(* IEC 61131-3 sources: Summary-ETFA22/benchmark/PLCopen_safety (part 2) *)

(* ---- SFOutControl.st ---- *)
PROGRAM Main
VAR_INPUT
    Activate : BOOL ;
    SSafeControl : SAFEBOOL ;
    ProcessControl : BOOL ;
    StaticControl : BOOL ;
    SStartReset : SAFEBOOL ;
    SAutoReset	: SAFEBOOL ;
    Reset : BOOL ;
END_VAR
VAR
    SFOutControl : SFOutControl;
END_VAR
SFOutControl(Activate:=Activate,SSafeControl:=SSafeControl,ProcessControl:=ProcessControl,StaticControl:=StaticControl,
SStartReset:=SStartReset,SAutoReset:=SAutoReset,Reset:=Reset);
END_PROGRAM

FUNCTION_BLOCK SFOutControl
VAR_INPUT
    Activate : BOOL ;
    SSafeControl : SAFEBOOL ;
    ProcessControl : BOOL ;
    StaticControl : BOOL ;
    SStartReset : SAFEBOOL ;
    SAutoReset	: SAFEBOOL ;
    Reset : BOOL ;
END_VAR
VAR
    RTRIGatResetQ : BOOL;
    RTRIGatResetM : BOOL;
    RTRIGatProcessControlQ : BOOL;
    RTRIGatProcessControlM : BOOL;
END_VAR
VAR_OUTPUT
    Ready : BOOL ;
    SOutControl : SAFEBOOL ;
    Error : BOOL ;
    DiagCode : WORD:=16#0000 ;
END_VAR
RTRIGatResetQ := Reset AND NOT RTRIGatResetM;
RTRIGatResetM := Reset;

RTRIGatProcessControlQ := ProcessControl AND NOT RTRIGatProcessControlM;
RTRIGatProcessControlM := ProcessControl;

IF NOT Activate THEN
    DiagCode := 16#0000;
ELSE
    CASE DiagCode OF
    16#0000:
        IF Activate THEN
            DiagCode := 16#8001;
        END_IF;
    16#8000:
        IF NOT SSafeControl THEN
            DiagCode := 16#8002;
        ELSIF NOT ProcessControl THEN
            DiagCode := 16#8010;
        END_IF;
    16#8001:
        IF Reset AND NOT RTRIGatResetQ AND NOT SStartReset THEN
            DiagCode := 16#C001;
        ELSIF RTRIGatResetQ AND RTRIGatProcessControlQ THEN
            DiagCode := 16#C111;
        ELSIF RTRIGatResetQ OR SStartReset THEN
            DiagCode := 16#8010;
        END_IF;
    16#8002:
        IF SSafeControl THEN
            DiagCode := 16#8003;
        END_IF;
    16#8003:
        IF NOT SSafeControl THEN
            DiagCode := 16#8002;
        ELSIF Reset AND NOT RTRIGatResetQ AND NOT SAutoReset THEN
            DiagCode := 16#C002;
        ELSIF RTRIGatResetQ AND RTRIGatProcessControlQ THEN
            DiagCode := 16#C211;
        ELSIF RTRIGatResetQ OR SAutoReset THEN
            DiagCode := 16#8010;
        END_IF;
    16#8010:
        IF NOT SSafeControl THEN
            DiagCode := 16#8002;
        ELSIF NOT RTRIGatProcessControlQ AND ProcessControl AND NOT StaticControl THEN
            DiagCode := 16#C010;
        ELSIF SSafeControl AND (RTRIGatProcessControlQ OR (StaticControl AND ProcessControl)) THEN
            DiagCode := 16#8000;
        END_IF;
    16#C001:
        IF NOT Reset THEN
            DiagCode := 16#8001;
        END_IF;
    16#C002:
        IF NOT Reset THEN
            DiagCode := 16#8003;
        END_IF;
    16#C010:
        IF NOT ProcessControl THEN
            DiagCode := 16#8010;
        END_IF;
    16#C111:
        IF NOT Reset THEN
            DiagCode := 16#8001;
        END_IF;
    16#C211:
        IF NOT Reset THEN
            DiagCode := 16#8003;
        END_IF;
    END_CASE;
END_IF;
CASE DiagCode OF
16#0000:
    Ready := FALSE;
    SOutControl := FALSE;
    Error := FALSE;
16#8000:
    Ready := TRUE;
    SOutControl := TRUE;
    Error := FALSE;
16#8001, 16#8002, 16#8003, 16#8010:
    Ready := TRUE;
    SOutControl := FALSE;
    Error := FALSE;
16#C001, 16#C002, 16#C010, 16#C111, 16#C211:
    Ready := TRUE;
    SOutControl := FALSE;
    Error := TRUE;
END_CASE;
END_FUNCTION_BLOCK

(* ---- SFOutControl_CAP.st ---- *)
PROGRAM Main
VAR_INPUT
    Activate : BOOL ;
    SSafeControl : SAFEBOOL ;
    ProcessControl : BOOL ;
    StaticControl : BOOL ;
    SStartReset : SAFEBOOL ;
    SAutoReset	: SAFEBOOL ;
    Reset : BOOL ;
END_VAR
VAR
    SFOutControl : SFOutControl;
END_VAR
SFOutControl(Activate:=Activate,SSafeControl:=SSafeControl,ProcessControl:=ProcessControl,StaticControl:=StaticControl,
SStartReset:=SStartReset,SAutoReset:=SAutoReset,Reset:=Reset);
END_PROGRAM

FUNCTION_BLOCK SFOutControl
VAR_INPUT
    Activate : BOOL ;
    SSafeControl : SAFEBOOL ;
    ProcessControl : BOOL ;
    StaticControl : BOOL ;
    SStartReset : SAFEBOOL ;
    SAutoReset	: SAFEBOOL ;
    Reset : BOOL ;
END_VAR
VAR
    RTRIGatResetQ : BOOL;
    RTRIGatResetM : BOOL;
    RTRIGatProcessControlQ : BOOL;
    RTRIGatProcessControlM : BOOL;
END_VAR
VAR_OUTPUT
    Ready : BOOL ;
    SOutControl : SAFEBOOL ;
    Error : BOOL ;
    DiagCode : WORD:=16#0000 ;
END_VAR
RTRIGatResetQ := Reset AND NOT RTRIGatResetM;
RTRIGatResetM := Reset;

RTRIGatProcessControlQ := ProcessControl AND NOT RTRIGatProcessControlM;
RTRIGatProcessControlM := ProcessControl;

IF NOT Activate THEN
    DiagCode := change(16#0000, 16#0000);
ELSE
    CASE DiagCode OF
    16#0000:
        IF Activate THEN
            DiagCode := 16#8001;
        END_IF;
    16#8000:
        IF NOT SSafeControl THEN
            DiagCode := 16#8002;
        ELSIF NOT ProcessControl THEN
            DiagCode := 16#8010;
        END_IF;
    16#8001:
        IF Reset AND NOT RTRIGatResetQ AND NOT SStartReset THEN
            DiagCode := 16#C001;
        ELSIF RTRIGatResetQ AND RTRIGatProcessControlQ THEN
            DiagCode := 16#C111;
        ELSIF RTRIGatResetQ OR SStartReset THEN
            DiagCode := 16#8010;
        END_IF;
    16#8002:
        IF SSafeControl THEN
            DiagCode := 16#8003;
        END_IF;
    16#8003:
        IF NOT SSafeControl THEN
            DiagCode := 16#8002;
        ELSIF Reset AND NOT RTRIGatResetQ AND NOT SAutoReset THEN
            DiagCode := 16#C002;
        ELSIF RTRIGatResetQ AND RTRIGatProcessControlQ THEN
            DiagCode := 16#C211;
        ELSIF RTRIGatResetQ OR SAutoReset THEN
            DiagCode := 16#8010;
        END_IF;
    16#8010:
        IF NOT SSafeControl THEN
            DiagCode := 16#8002;
        ELSIF NOT RTRIGatProcessControlQ AND ProcessControl AND NOT StaticControl THEN
            DiagCode := 16#C010;
        ELSIF SSafeControl AND (RTRIGatProcessControlQ OR (StaticControl AND ProcessControl)) THEN
            DiagCode := 16#8000;
        END_IF;
    16#C001:
        IF NOT Reset THEN
            DiagCode := change(16#8001, 16#C002);
        END_IF;
    16#C002:
        IF NOT Reset THEN
            DiagCode := 16#8003;
        END_IF;
    16#C010:
        IF NOT ProcessControl THEN
            DiagCode := 16#8010;
        END_IF;
    16#C111:
        IF NOT Reset THEN
            DiagCode := 16#8001;
        END_IF;
    16#C211:
        IF NOT Reset THEN
            DiagCode := 16#8003;
        END_IF;
    END_CASE;
END_IF;
CASE DiagCode OF
16#0000:
    Ready := FALSE;
    SOutControl := FALSE;
    Error := FALSE;
16#8000:
    Ready := TRUE;
    SOutControl := TRUE;
    Error := FALSE;
16#8001, 16#8002, 16#8003, 16#8010:
    Ready := TRUE;
    SOutControl := FALSE;
    Error := FALSE;
16#C001, 16#C002, 16#C010, 16#C111, 16#C211:
    Ready := TRUE;
    SOutControl := FALSE;
    Error := TRUE;
END_CASE;
END_FUNCTION_BLOCK

(* ---- SFSafelyLimitSpeed.st ---- *)
PROGRAM Main
VAR_INPUT
    Activate : BOOL;
    SOpMode : SAFEBOOL;
    SEnabled : SAFEBOOL;
    AxisID : INT;
    MonitoringTime : TIME;
    Reset : BOOL;
    Acknowledge : BOOL;      (* This is an internal input *)
END_VAR
VAR
    SFSafelyLimitSpeed : SFSafelyLimitSpeed;
END_VAR
SFSafelyLimitSpeed(Activate:=Activate,SOpMode:=SOpMode,SEnabled:=SEnabled,AxisID:=AxisID,MonitoringTime:=MonitoringTime,
Reset:=Reset,Acknowledge:=Acknowledge);
END_PROGRAM

FUNCTION_BLOCK SFSafelyLimitSpeed
VAR_INPUT
    Activate : BOOL;
    SOpMode : SAFEBOOL;
    SEnabled : SAFEBOOL;
    AxisID : INT;
    MonitoringTime : TIME;
    Reset : BOOL;
    Acknowledge : BOOL;      (* This is an internal input *)
END_VAR
VAR
    IN : BOOL;
    PT : TIME;
    running : BOOL;
    Q : BOOL;
    RTRIGatResetQ : BOOL;
    RTRIGatResetM : BOOL;
END_VAR
VAR_OUTPUT
    Ready : BOOL;
    SSafetyActive : SAFEBOOL;
    Error : BOOL;
    DiagCode : WORD;
END_VAR
RTRIGatResetQ := Reset AND NOT RTRIGatResetM;
RTRIGatResetM := Reset;

IF NOT Activate THEN
    DiagCode := 16#0000;
END_IF;
IN:=Activate AND NOT SOpMode;
PT:=MonitoringTime;
IF NOT IN THEN
    Q := FALSE;
    running := FALSE;
ELSIF NOT running AND NOT Q THEN
    running := TRUE;
ELSIF running AND NOT Q THEN
    Q := NONDETERMINISTIC_BOOL();
    running := NOT Q;
END_IF;
CASE DiagCode OF
16#0000:
    IF Activate THEN
        DiagCode := 16#8001;
    END_IF;
16#8000:
    IF NOT Acknowledge THEN
        DiagCode := 16#C002;
    ELSIF SOpMode THEN
        DiagCode := 16#8012;
    ELSIF SEnabled THEN
        DiagCode := 16#8004;
    END_IF;
16#8001:
    IF Reset AND NOT RTRIGatResetQ THEN
        DiagCode := 16#C001;
    ELSIF RTRIGatResetQ AND NOT Acknowledge THEN
        DiagCode := 16#8002;
    ELSIF RTRIGatResetQ AND Acknowledge THEN
        DiagCode := 16#8012;
    END_IF;
16#8002:
    IF NOT SOpMode THEN
        DiagCode := 16#8003;
    ELSIF Acknowledge THEN
        DiagCode := 16#8012;
    END_IF;
16#8003:
    IF Q THEN
        DiagCode := 16#C003;
    ELSIF SOpMode THEN
        DiagCode := 16#8012;
    ELSIF Acknowledge AND NOT SEnabled THEN
        DiagCode := 16#8000;
    ELSIF Acknowledge AND SEnabled THEN
        DiagCode := 16#8004;
    END_IF;
16#8004:
    IF NOT Acknowledge THEN
        DiagCode := 16#C002;
    ELSIF SOpMode THEN
        DiagCode := 16#8012;
    ELSIF NOT SEnabled THEN
        DiagCode := 16#8000;
    END_IF;
16#8005:
    IF SOpMode THEN
        DiagCode := 16#8012;
    END_IF;
16#8012:
    IF NOT Acknowledge THEN
        DiagCode := 16#8002;
    ELSIF NOT SOpMode THEN
        DiagCode := 16#8003;
    END_IF;
16#C001:
    IF NOT Reset THEN
        DiagCode := 16#8001;
    END_IF;
16#C002:
    IF Reset AND NOT RTRIGatResetQ THEN
        DiagCode := 16#C004;
    ELSIF RTRIGatResetQ THEN
        DiagCode := 16#8005;
    END_IF;
16#C003:
    IF Reset AND NOT RTRIGatResetQ THEN
        DiagCode := 16#C005;
    ELSIF RTRIGatResetQ THEN
        DiagCode := 16#8005;
    END_IF;
16#C004:
    IF NOT Reset THEN
        DiagCode := 16#C002;
    END_IF;
16#C005:
    IF NOT Reset THEN
        DiagCode := 16#C003;
    END_IF;
END_CASE;
CASE DiagCode OF
16#0000:
    Ready := FALSE;
    SSafetyActive := FALSE;
    Error := FALSE;
16#8000,
16#8004:
    Ready := TRUE;
    SSafetyActive := TRUE;
    Error := FALSE;
16#8001,
16#8002,
16#8003,
16#8005,
16#8012:
    Ready := TRUE;
    SSafetyActive := FALSE;
    Error := FALSE;
16#C001,
16#C002,
16#C003,
16#C004,
16#C005:
    Ready := TRUE;
    SSafetyActive := FALSE;
    Error := TRUE;
END_CASE;
END_FUNCTION_BLOCK

(* ---- SFSafelyLimitSpeed_CAP.st ---- *)
PROGRAM Main
VAR_INPUT
    Activate : BOOL;
    SOpMode : SAFEBOOL;
    SEnabled : SAFEBOOL;
    AxisID : INT;
    MonitoringTime : TIME;
    Reset : BOOL;
    Acknowledge : BOOL;      (* This is an internal input *)
END_VAR
VAR
    SFSafelyLimitSpeed : SFSafelyLimitSpeed;
END_VAR
SFSafelyLimitSpeed(Activate:=Activate,SOpMode:=SOpMode,SEnabled:=SEnabled,AxisID:=AxisID,MonitoringTime:=MonitoringTime,
Reset:=Reset,Acknowledge:=Acknowledge);
END_PROGRAM

FUNCTION_BLOCK SFSafelyLimitSpeed
VAR_INPUT
    Activate : BOOL;
    SOpMode : SAFEBOOL;
    SEnabled : SAFEBOOL;
    AxisID : INT;
    MonitoringTime : TIME;
    Reset : BOOL;
    Acknowledge : BOOL;      (* This is an internal input *)
END_VAR
VAR
    IN : BOOL;
    PT : TIME;
    running : BOOL;
    Q : BOOL;
    RTRIGatResetQ : BOOL;
    RTRIGatResetM : BOOL;
END_VAR
VAR_OUTPUT
    Ready : BOOL;
    SSafetyActive : SAFEBOOL;
    Error : BOOL;
    DiagCode : WORD;
END_VAR
RTRIGatResetQ := Reset AND NOT RTRIGatResetM;
RTRIGatResetM := Reset;

IF NOT Activate THEN
    DiagCode := 16#0000;
END_IF;
IN:=Activate AND NOT SOpMode;
PT:=MonitoringTime;
IF NOT IN THEN
    Q := FALSE;
    running := FALSE;
ELSIF NOT running AND NOT Q THEN
    running := TRUE;
ELSIF running AND NOT Q THEN
    Q := NONDETERMINISTIC_BOOL();
    running := NOT Q;
END_IF;
CASE DiagCode OF
16#0000:
    IF Activate THEN
        DiagCode := 16#8001;
    END_IF;
16#8000:
    IF NOT Acknowledge THEN
        DiagCode := change(16#C002, 16#8012);
    ELSIF SOpMode THEN
        DiagCode := 16#8012;
    ELSIF SEnabled THEN
        DiagCode := 16#8004;
    END_IF;
16#8001:
    IF Reset AND NOT RTRIGatResetQ THEN
        DiagCode := 16#C001;
    ELSIF RTRIGatResetQ AND NOT Acknowledge THEN
        DiagCode := 16#8002;
    ELSIF RTRIGatResetQ AND Acknowledge THEN
        DiagCode := 16#8012;
    END_IF;
16#8002:
    IF NOT SOpMode THEN
        DiagCode := 16#8003;
    ELSIF Acknowledge THEN
        DiagCode := 16#8012;
    END_IF;
16#8003:
    IF Q THEN
        DiagCode := 16#C003;
    ELSIF SOpMode THEN
        DiagCode := 16#8012;
    ELSIF Acknowledge AND NOT SEnabled THEN
        DiagCode := 16#8000;
    ELSIF Acknowledge AND SEnabled THEN
        DiagCode := 16#8004;
    END_IF;
16#8004:
    IF NOT Acknowledge THEN
        DiagCode := 16#C002;
    ELSIF SOpMode THEN
        DiagCode := 16#8012;
    ELSIF NOT SEnabled THEN
        DiagCode := 16#8000;
    END_IF;
16#8005:
    IF SOpMode THEN
        DiagCode := 16#8012;
    END_IF;
16#8012:
    IF NOT Acknowledge THEN
        DiagCode := 16#8002;
    ELSIF NOT SOpMode THEN
        DiagCode := 16#8003;
    END_IF;
16#C001:
    IF NOT Reset THEN
        DiagCode := 16#8001;
    END_IF;
16#C002:
    IF Reset AND NOT RTRIGatResetQ THEN
        DiagCode := 16#C004;
    ELSIF RTRIGatResetQ THEN
        DiagCode := 16#8005;
    END_IF;
16#C003:
    IF Reset AND NOT RTRIGatResetQ THEN
        DiagCode := 16#C005;
    ELSIF RTRIGatResetQ THEN
        DiagCode := 16#8005;
    END_IF;
16#C004:
    IF NOT Reset THEN
        DiagCode := 16#C002;
    END_IF;
16#C005:
    IF NOT Reset THEN
        DiagCode := 16#C003;
    END_IF;
END_CASE;
CASE DiagCode OF
16#0000:
    Ready := FALSE;
    SSafetyActive := FALSE;
    Error := FALSE;
16#8000,
16#8004:
    Ready := TRUE;
    SSafetyActive := TRUE;
    Error := FALSE;
16#8001,
16#8002,
16#8003,
16#8005,
16#8012:
    Ready := TRUE;
    SSafetyActive := FALSE;
    Error := FALSE;
16#C001,
16#C002,
16#C003,
16#C004,
16#C005:
    Ready := TRUE;
    SSafetyActive := FALSE;
    Error := TRUE;
END_CASE;
END_FUNCTION_BLOCK

(* ---- SFSafeStop.st ---- *)
PROGRAM Main
VAR_INPUT
    Activate : BOOL;
    SStopIn : SAFEBOOL;
    AxisID : INT;
    MonitoringTime : TIME;
    Reset : BOOL;
    Acknowledge : BOOL;      (* This is an internal input *)
END_VAR
VAR
    SFSafeStop : SFSafeStop;
END_VAR
SFSafeStop(Activate:=Activate,SStopIn:=SStopIn,AxisID:=AxisID,MonitoringTime:=MonitoringTime,Reset:=Reset,
Acknowledge:=Acknowledge);
END_PROGRAM

FUNCTION_BLOCK SFSafeStop
VAR_INPUT
    Activate : BOOL;
    SStopIn : SAFEBOOL;
    AxisID : INT;
    MonitoringTime : TIME;
    Reset : BOOL;
    Acknowledge : BOOL;      (* This is an internal input *)
END_VAR
VAR
    IN : BOOL;
    PT : TIME;
    running : BOOL;
    Q : BOOL;
    RTRIGatResetQ : BOOL;
    RTRIGatResetM : BOOL;
END_VAR
VAR_OUTPUT
    Ready : BOOL;
    SStopped : SAFEBOOL;
    Error : BOOL;
    DiagCode : WORD:=16#0000;
END_VAR
RTRIGatResetQ := Reset AND NOT RTRIGatResetM;
RTRIGatResetM := Reset;
IF NOT Activate THEN
    DiagCode := 16#0000;
ELSE
    IN:=Activate AND NOT SStopIn;
    PT:=MonitoringTime;
    IF NOT IN THEN
        Q := FALSE;
        running := FALSE;
    ELSIF NOT running AND NOT Q THEN
        running := TRUE;
    ELSIF running AND NOT Q THEN
        Q := NONDETERMINISTIC_BOOL();
        running := NOT Q;
    END_IF;
    CASE DiagCode OF
    16#0000:
        IF Activate THEN
            DiagCode := 16#8001;
        END_IF;
    16#8000:
        IF NOT Acknowledge THEN
            DiagCode := 16#C002;
        ELSIF SStopIn THEN
            DiagCode := 16#8012;
        END_IF;
    16#8001:
        IF RTRIGatResetQ AND NOT Acknowledge THEN
            DiagCode := 16#8002;
        ELSIF RTRIGatResetQ AND Acknowledge THEN
            DiagCode := 16#8012;
        END_IF;
    16#8002:
        IF NOT SStopIn THEN
            DiagCode := 16#8003;
        ELSIF Acknowledge THEN
            DiagCode := 16#8012;
        END_IF;
    16#8003:
        IF Q THEN
            DiagCode := 16#C003;
        ELSIF SStopIn THEN
            DiagCode := 16#8012;
        ELSIF Acknowledge THEN
            DiagCode := 16#8000;
        END_IF;
    16#8005:
        IF SStopIn THEN
            DiagCode := 16#8012;
        END_IF;
    16#8012:
        IF NOT Acknowledge THEN
            DiagCode := 16#8002;
        ELSIF NOT SStopIn THEN
            DiagCode := 16#8003;
        ELSIF Acknowledge THEN
            DiagCode := 16#8000;
        END_IF;
    16#C002:
        IF Reset AND NOT RTRIGatResetQ THEN
            DiagCode := 16#C004;
        ELSIF RTRIGatResetQ THEN
            DiagCode := 16#8005;
        END_IF;
    16#C003:
        IF Reset AND NOT RTRIGatResetQ THEN
            DiagCode := 16#C005;
        ELSIF RTRIGatResetQ THEN
            DiagCode := 16#8005;
        END_IF;
    16#C004:
        IF NOT Reset THEN
            DiagCode := 16#C002;
        END_IF;
    16#C005:
        IF NOT Reset THEN
            DiagCode := 16#C003;
        END_IF;
    END_CASE;
END_IF;
CASE DiagCode OF
16#0000:
    Ready := FALSE;
    SStopped := FALSE;
    Error := FALSE;
16#8000:
    Ready := TRUE;
    SStopped := TRUE;
    Error := FALSE;
16#8001,
16#8002,
16#8003,
16#8005,
16#8012:
    Ready := TRUE;
    SStopped := FALSE;
    Error := FALSE;
16#C002,
16#C003,
16#C004,
16#C005:
    Ready := TRUE;
    SStopped := FALSE;
    Error := TRUE;
END_CASE;
END_FUNCTION_BLOCK

(* ---- SFSafeStop_CAP.st ---- *)
PROGRAM Main
VAR_INPUT
    Activate : BOOL;
    SStopIn : SAFEBOOL;
    AxisID : INT;
    MonitoringTime : TIME;
    Reset : BOOL;
    Acknowledge : BOOL;      (* This is an internal input *)
END_VAR
VAR
    SFSafeStop : SFSafeStop;
END_VAR
SFSafeStop(Activate:=Activate,SStopIn:=SStopIn,AxisID:=AxisID,MonitoringTime:=MonitoringTime,Reset:=Reset,
Acknowledge:=Acknowledge);
END_PROGRAM

FUNCTION_BLOCK SFSafeStop
VAR_INPUT
    Activate : BOOL;
    SStopIn : SAFEBOOL;
    AxisID : INT;
    MonitoringTime : TIME;
    Reset : BOOL;
    Acknowledge : BOOL;      (* This is an internal input *)
END_VAR
VAR
    IN : BOOL;
    PT : TIME;
    running : BOOL;
    Q : BOOL;
    RTRIGatResetQ : BOOL;
    RTRIGatResetM : BOOL;
END_VAR
VAR_OUTPUT
    Ready : BOOL;
    SStopped : SAFEBOOL;
    Error : BOOL;
    DiagCode : WORD:=16#0000;
END_VAR
RTRIGatResetQ := Reset AND NOT RTRIGatResetM;
RTRIGatResetM := Reset;
IF NOT Activate THEN
    DiagCode := 16#0000;
ELSE
    IN:=Activate AND NOT SStopIn;
    PT:=MonitoringTime;
    IF NOT IN THEN
        Q := FALSE;
        running := FALSE;
    ELSIF NOT running AND NOT Q THEN
        running := TRUE;
    ELSIF running AND NOT Q THEN
        Q := NONDETERMINISTIC_BOOL();
        running := NOT Q;
    END_IF;
    CASE DiagCode OF
    16#0000:
        IF Activate THEN
            DiagCode := change(16#8001, 16#8000);
        END_IF;
    16#8000:
        IF NOT Acknowledge THEN
            DiagCode := 16#C002;
        ELSIF SStopIn THEN
            DiagCode := 16#8012;
        END_IF;
    16#8001:
        IF RTRIGatResetQ AND NOT Acknowledge THEN
            DiagCode := 16#8002;
        ELSIF RTRIGatResetQ AND Acknowledge THEN
            DiagCode := 16#8012;
        END_IF;
    16#8002:
        IF NOT SStopIn THEN
            DiagCode := 16#8003;
        ELSIF Acknowledge THEN
            DiagCode := 16#8012;
        END_IF;
    16#8003:
        IF Q THEN
            DiagCode := 16#C003;
        ELSIF SStopIn THEN
            DiagCode := 16#8012;
        ELSIF Acknowledge THEN
            DiagCode := 16#8000;
        END_IF;
    16#8005:
        IF SStopIn THEN
            DiagCode := 16#8012;
        END_IF;
    16#8012:
        IF NOT Acknowledge THEN
            DiagCode := 16#8002;
        ELSIF NOT SStopIn THEN
            DiagCode := 16#8003;
        ELSIF Acknowledge THEN
            DiagCode := 16#8000;
        END_IF;
    16#C002:
        IF Reset AND NOT RTRIGatResetQ THEN
            DiagCode := 16#C004;
        ELSIF RTRIGatResetQ THEN
            DiagCode := 16#8005;
        END_IF;
    16#C003:
        IF Reset AND NOT RTRIGatResetQ THEN
            DiagCode := 16#C005;
        ELSIF RTRIGatResetQ THEN
            DiagCode := 16#8005;
        END_IF;
    16#C004:
        IF NOT Reset THEN
            DiagCode := 16#C002;
        END_IF;
    16#C005:
        IF NOT Reset THEN
            DiagCode := 16#C003;
        END_IF;
    END_CASE;
END_IF;
CASE DiagCode OF
16#0000:
    Ready := FALSE;
    SStopped := FALSE;
    Error := FALSE;
16#8000:
    Ready := TRUE;
    SStopped := TRUE;
    Error := FALSE;
16#8001,
16#8002,
16#8003,
16#8005,
16#8012:
    Ready := TRUE;
    SStopped := FALSE;
    Error := FALSE;
16#C002,
16#C003,
16#C004,
16#C005:
    Ready := TRUE;
    SStopped := FALSE;
    Error := TRUE;
END_CASE;
END_FUNCTION_BLOCK

(* ---- SFSafetyRequest.st ---- *)
PROGRAM Main
VAR_INPUT
    Activate : BOOL;
    SOpMode : SAFEBOOL;
    SAcknowledge : SAFEBOOL;
    MonitoringTime : TIME;
    Reset : BOOL;
END_VAR
VAR
    SFSafetyRequest : SFSafetyRequest;
END_VAR
SFSafetyRequest(Activate:=Activate,SOpMode:=SOpMode,SAcknowledge:=SAcknowledge,MonitoringTime:=MonitoringTime,Reset:=Reset);
END_PROGRAM

FUNCTION_BLOCK SFSafetyRequest
VAR_INPUT
    Activate : BOOL;
    SOpMode : SAFEBOOL;
    SAcknowledge : SAFEBOOL;
    MonitoringTime : TIME;
    Reset : BOOL;
END_VAR
VAR
    RTRIGatResetQ : BOOL;
    RTRIGatResetM : BOOL;
    IN : BOOL;
    PT : TIME;
    running : BOOL;
    Q : BOOL;
END_VAR
VAR_OUTPUT
    Ready : BOOL;
    SSafetyActive : SAFEBOOL;
    SSafetyRequest : SAFEBOOL;
    Error : BOOL;
    DiagCode : WORD;
END_VAR
RTRIGatResetQ := Reset AND NOT RTRIGatResetM;
RTRIGatResetM := Reset;

IF NOT Activate THEN
    DiagCode := 16#0000;
ELSE
    CASE DiagCode OF
    16#0000:
        IF Activate THEN
            DiagCode := 16#8001;
        END_IF;
    16#8000:
        IF NOT SAcknowledge THEN
            DiagCode := 16#C002;
        ELSIF SOpMode THEN
            DiagCode := 16#8012;
        END_IF;
    16#8001:
        IF RTRIGatResetQ AND NOT SAcknowledge THEN
            DiagCode := 16#8002;
        ELSIF RTRIGatResetQ AND SAcknowledge THEN
            DiagCode := 16#8012;
        END_IF;
    16#8002:
        IF NOT SOpMode THEN
            DiagCode := 16#8003;
        ELSIF SAcknowledge THEN
            DiagCode := 16#8012;
        END_IF;
    16#8003:
        IF Q THEN
            DiagCode := 16#C003;
        ELSIF SOpMode THEN
            DiagCode := 16#8012;
        ELSIF SAcknowledge THEN
            DiagCode := 16#8000;
        END_IF;
    16#8005:
        IF SOpMode THEN
            DiagCode := 16#8012;
        END_IF;
    16#8012:
        IF NOT SAcknowledge THEN
            DiagCode := 16#8002;
        ELSIF NOT SOpMode THEN
            DiagCode := 16#8003;
        END_IF;
    16#C002:
        IF Reset AND NOT RTRIGatResetQ THEN
            DiagCode := 16#C004;
        ELSIF RTRIGatResetQ THEN
            DiagCode := 16#8005;
        END_IF;
    16#C003:
        IF Reset AND NOT RTRIGatResetQ THEN
            DiagCode := 16#C005;
        ELSIF RTRIGatResetQ THEN
            DiagCode := 16#8005;
        END_IF;
    16#C004:
        IF NOT Reset THEN
            DiagCode := 16#C002;
        END_IF;
    16#C005:
        IF NOT Reset THEN
            DiagCode := 16#C003;
        END_IF;
    END_CASE;
END_IF;
IF DiagCode <> 16#8003 THEN
    IN:=FALSE;
    PT:=MonitoringTime;
    Q := FALSE;
    running := FALSE;
ELSE
    IN:=TRUE;
    PT:=MonitoringTime;
    IF NOT running AND NOT Q THEN
        running := TRUE;
    ELSIF running AND NOT Q THEN
        Q := NONDETERMINISTIC_BOOL();
        running := NOT Q;
    END_IF;
END_IF;
CASE DiagCode OF
16#0000:
    Ready := FALSE;
    SSafetyActive := FALSE;
    SSafetyRequest := FALSE;
    Error := FALSE;
16#8000:
    Ready := TRUE;
    SSafetyActive := TRUE;
    SSafetyRequest := FALSE;
    Error := FALSE;
16#8001:
    Ready := TRUE;
    SSafetyActive := FALSE;
    SSafetyRequest := FALSE;
    Error := FALSE;
16#8002:
    Ready := TRUE;
    SSafetyActive := FALSE;
    SSafetyRequest := TRUE;
    Error := FALSE;
16#8003:
    Ready := TRUE;
    SSafetyActive := FALSE;
    SSafetyRequest := FALSE;
    Error := FALSE;
16#8005:
    Ready := TRUE;
    SSafetyActive := FALSE;
    SSafetyRequest := FALSE;
    Error := FALSE;
16#8012:
    Ready := TRUE;
    SSafetyActive := FALSE;
    SSafetyRequest := TRUE;
    Error := FALSE;
16#C002:
    Ready := TRUE;
    SSafetyActive := FALSE;
    SSafetyRequest := FALSE;
    Error := TRUE;
16#C003:
    Ready := TRUE;
    SSafetyActive := FALSE;
    SSafetyRequest := FALSE;
    Error := TRUE;
16#C004:
    Ready := TRUE;
    SSafetyActive := FALSE;
    SSafetyRequest := FALSE;
    Error := TRUE;
16#C005:
    Ready := TRUE;
    SSafetyActive := FALSE;
    SSafetyRequest := FALSE;
    Error := TRUE;
END_CASE;
END_FUNCTION_BLOCK

(* ---- SFSafetyRequest_CAP.st ---- *)
PROGRAM Main
VAR_INPUT
    Activate : BOOL;
    SOpMode : SAFEBOOL;
    SAcknowledge : SAFEBOOL;
    MonitoringTime : TIME;
    Reset : BOOL;
END_VAR
VAR
    SFSafetyRequest : SFSafetyRequest;
END_VAR
SFSafetyRequest(Activate:=Activate,SOpMode:=SOpMode,SAcknowledge:=SAcknowledge,MonitoringTime:=MonitoringTime,Reset:=Reset);
END_PROGRAM

FUNCTION_BLOCK SFSafetyRequest
VAR_INPUT
    Activate : BOOL;
    SOpMode : SAFEBOOL;
    SAcknowledge : SAFEBOOL;
    MonitoringTime : TIME;
    Reset : BOOL;
END_VAR
VAR
    RTRIGatResetQ : BOOL;
    RTRIGatResetM : BOOL;
    IN : BOOL;
    PT : TIME;
    running : BOOL;
    Q : BOOL;
END_VAR
VAR_OUTPUT
    Ready : BOOL;
    SSafetyActive : SAFEBOOL;
    SSafetyRequest : SAFEBOOL;
    Error : BOOL;
    DiagCode : WORD;
END_VAR
RTRIGatResetQ := Reset AND NOT RTRIGatResetM;
RTRIGatResetM := Reset;

IF NOT Activate THEN
    DiagCode := 16#0000;
ELSE
    CASE DiagCode OF
    16#0000:
        IF Activate THEN
            DiagCode := 16#8001;
        END_IF;
    16#8000:
        IF NOT SAcknowledge THEN
            DiagCode := 16#C002;
        ELSIF SOpMode THEN
            DiagCode := change(16#8012, 16#8003);
        END_IF;
    16#8001:
        IF RTRIGatResetQ AND NOT SAcknowledge THEN
            DiagCode := 16#8002;
        ELSIF RTRIGatResetQ AND SAcknowledge THEN
            DiagCode := 16#8012;
        END_IF;
    16#8002:
        IF NOT SOpMode THEN
            DiagCode := 16#8003;
        ELSIF SAcknowledge THEN
            DiagCode := 16#8012;
        END_IF;
    16#8003:
        IF Q THEN
            DiagCode := 16#C003;
        ELSIF SOpMode THEN
            DiagCode := 16#8012;
        ELSIF SAcknowledge THEN
            DiagCode := 16#8000;
        END_IF;
    16#8005:
        IF SOpMode THEN
            DiagCode := 16#8012;
        END_IF;
    16#8012:
        IF NOT SAcknowledge THEN
            DiagCode := 16#8002;
        ELSIF NOT SOpMode THEN
            DiagCode := 16#8003;
        END_IF;
    16#C002:
        IF Reset AND NOT RTRIGatResetQ THEN
            DiagCode := 16#C004;
        ELSIF RTRIGatResetQ THEN
            DiagCode := 16#8005;
        END_IF;
    16#C003:
        IF Reset AND NOT RTRIGatResetQ THEN
            DiagCode := 16#C005;
        ELSIF RTRIGatResetQ THEN
            DiagCode := 16#8005;
        END_IF;
    16#C004:
        IF NOT Reset THEN
            DiagCode := 16#C002;
        END_IF;
    16#C005:
        IF NOT Reset THEN
            DiagCode := 16#C003;
        END_IF;
    END_CASE;
END_IF;
IF DiagCode <> 16#8003 THEN
    IN:=FALSE;
    PT:=MonitoringTime;
    Q := FALSE;
    running := FALSE;
ELSE
    IN:=TRUE;
    PT:=MonitoringTime;
    IF NOT running AND NOT Q THEN
        running := TRUE;
    ELSIF running AND NOT Q THEN
        Q := NONDETERMINISTIC_BOOL();
        running := NOT Q;
    END_IF;
END_IF;
CASE DiagCode OF
16#0000:
    Ready := FALSE;
    SSafetyActive := FALSE;
    SSafetyRequest := FALSE;
    Error := FALSE;
16#8000:
    Ready := TRUE;
    SSafetyActive := TRUE;
    SSafetyRequest := FALSE;
    Error := FALSE;
16#8001:
    Ready := TRUE;
    SSafetyActive := FALSE;
    SSafetyRequest := FALSE;
    Error := FALSE;
16#8002:
    Ready := TRUE;
    SSafetyActive := FALSE;
    SSafetyRequest := TRUE;
    Error := FALSE;
16#8003:
    Ready := TRUE;
    SSafetyActive := FALSE;
    SSafetyRequest := FALSE;
    Error := FALSE;
16#8005:
    Ready := TRUE;
    SSafetyActive := FALSE;
    SSafetyRequest := FALSE;
    Error := FALSE;
16#8012:
    Ready := TRUE;
    SSafetyActive := FALSE;
    SSafetyRequest := TRUE;
    Error := FALSE;
16#C002:
    Ready := TRUE;
    SSafetyActive := FALSE;
    SSafetyRequest := FALSE;
    Error := TRUE;
16#C003:
    Ready := TRUE;
    SSafetyActive := FALSE;
    SSafetyRequest := FALSE;
    Error := TRUE;
16#C004:
    Ready := TRUE;
    SSafetyActive := FALSE;
    SSafetyRequest := FALSE;
    Error := TRUE;
16#C005:
    Ready := TRUE;
    SSafetyActive := FALSE;
    SSafetyRequest := FALSE;
    Error := TRUE;
END_CASE;
END_FUNCTION_BLOCK

(* ---- SFTestableSafetySensor.st ---- *)
PROGRAM Main
VAR_INPUT
    Activate : BOOL;
    SOSSDIn : SAFEBOOL;
    StartTest : BOOL;
    TestTime : TIME := T#10ms;
    NoExternalTest : BOOL;
    SStartReset : SAFEBOOL;
    SAutoReset : SAFEBOOL;
    Reset : BOOL;
END_VAR
VAR
    SFTestableSafetySensor : SFTestableSafetySensor;
END_VAR
SFTestableSafetySensor(Activate:=Activate,SOSSDIn:=SOSSDIn,StartTest:=StartTest,TestTime:=TestTime,NoExternalTest:=NoExternalTest,
SStartReset:=SStartReset,SAutoReset:=SAutoReset,Reset:=Reset);
END_PROGRAM

FUNCTION_BLOCK SFTestableSafetySensor
VAR_INPUT
    Activate : BOOL;
    SOSSDIn : SAFEBOOL;
    StartTest : BOOL;
    TestTime : TIME := T#10ms;
    NoExternalTest : BOOL;
    SStartReset : SAFEBOOL;
    SAutoReset : SAFEBOOL;
    Reset : BOOL;
END_VAR
VAR
    IN1 : BOOL;
    PT1 : TIME;
    running1 : BOOL;
    Q1 : BOOL;
    IN2 : BOOL;
    PT2 : TIME;
    running2 : BOOL;
    Q2 : BOOL;
    RTRIGatResetQ : BOOL;
    RTRIGatResetM : BOOL;
    RTRIGatStartTestQ : BOOL;
    RTRIGatStartTestM : BOOL;
    FTRIGatSOSSDInQ : BOOL;
    FTRIGatSOSSDInM : BOOL;
END_VAR
VAR_OUTPUT
    Ready : SAFEBOOL;
    SOSSDOut : SAFEBOOL;
    STestOut : SAFEBOOL := TRUE;
    TestPossible : BOOL;
    TestExecuted : BOOL;
    Error : BOOL;
    DiagCode : WORD := 16#0000;
END_VAR
RTRIGatResetQ := Reset AND NOT RTRIGatResetM;
RTRIGatResetM := Reset;

RTRIGatStartTestQ := StartTest AND NOT RTRIGatStartTestM;
RTRIGatStartTestM := StartTest;

FTRIGatSOSSDInQ := NOT SOSSDIn AND FTRIGatSOSSDInM;
FTRIGatSOSSDInM := SOSSDIn;

IF NOT Activate THEN
    DiagCode := 16#0000;
ELSE
    CASE DiagCode OF
    16#0000:
        IF Activate THEN
            DiagCode := 16#8001;
        END_IF;
    16#8000:
        IF NOT SOSSDIn THEN
            DiagCode := 16#8012;
        ELSIF RTRIGatStartTestQ THEN
            DiagCode := 16#8020;
            IN1:=FALSE;
            Q1 := FALSE;
            running1 := FALSE;
        END_IF;
    16#8001:
        IF TestTime > T#150ms THEN
            DiagCode := 16#C000;
        ELSIF Reset AND NOT RTRIGatResetQ AND NOT SStartReset THEN
            DiagCode := 16#C001;
        ELSIF NOT SOSSDIn THEN
            DiagCode := 16#8002;
        ELSIF SOSSDIn AND (RTRIGatResetQ OR SStartReset) THEN
            DiagCode := 16#8010;
        END_IF;
    16#8002:
        IF SOSSDIn THEN
            DiagCode := 16#8003;
        END_IF;
    16#8003:
        IF Reset AND NOT RTRIGatResetQ AND NOT SAutoReset THEN
            DiagCode := 16#C002;
        ELSIF NOT SOSSDIn THEN
            DiagCode := 16#8002;
        ELSIF SOSSDIn AND (RTRIGatResetQ OR SAutoReset) THEN
            DiagCode := 16#8010;
        END_IF;
    16#8004:
        IF FTRIGatSOSSDInQ THEN
            DiagCode := 16#8005;
        END_IF;
    16#8005:
        IF SOSSDIn THEN
            DiagCode := 16#8006;
        END_IF;
    16#8006:
        IF Reset AND NOT RTRIGatResetQ THEN
            DiagCode := 16#C005;
        ELSIF RTRIGatResetQ AND NOT SOSSDIn THEN
            DiagCode := 16#8002;
        ELSIF RTRIGatResetQ AND SOSSDIn THEN
            DiagCode := 16#8010;
        END_IF;
    16#8010:
        IF NOT SOSSDIn THEN
            DiagCode := 16#8002;
        ELSIF RTRIGatStartTestQ THEN
            DiagCode := 16#8020;
            IN1:=FALSE;
            Q1 := FALSE;
            running1 := FALSE;
        END_IF;
    16#8012:
        IF SOSSDIn THEN
            DiagCode := 16#8013;
        END_IF;
    16#8013:
        IF Reset AND NOT RTRIGatResetQ AND NOT SAutoReset THEN
            DiagCode := 16#C007;
        ELSIF NOT SOSSDIn THEN
            DiagCode := 16#8012;
        ELSIF SOSSDIn AND (RTRIGatResetQ OR SAutoReset) THEN
            DiagCode := 16#8000;
        END_IF;
    16#8020:
        IF Q1 THEN
            DiagCode := 16#C020;
        ELSIF NOT SOSSDIn THEN
            DiagCode := 16#8030;
            IN2:=FALSE;
            Q2 := FALSE;
            running2 := FALSE;
        END_IF;
    16#8030:
        IF Q2 THEN
            DiagCode := 16#C030;
        ELSIF SOSSDIn THEN
            DiagCode := 16#8000;
        END_IF;
    16#C000:
        IF Reset AND NOT RTRIGatResetQ THEN
            DiagCode := 16#C006;
        ELSIF RTRIGatResetQ AND TestTime <= T#150ms THEN
            DiagCode := 16#8001;
        END_IF;
    16#C001:
        IF NOT Reset THEN
            DiagCode := 16#8001;
        END_IF;
    16#C002:
        IF NOT Reset THEN
            DiagCode := 16#8003;
        END_IF;
    16#C003:
        IF NOT Reset THEN
            DiagCode := 16#C010;
        END_IF;
    16#C004:
        IF NOT Reset THEN
            DiagCode := 16#C020;
        END_IF;
    16#C005:
        IF NOT Reset THEN
            DiagCode := 16#8006;
        END_IF;
    16#C006:
        IF NOT Reset THEN
            DiagCode := 16#C000;
        END_IF;
    16#C007:
        IF NOT Reset THEN
            DiagCode := 16#8013;
        END_IF;
    16#C010:
        IF Reset AND NOT RTRIGatResetQ THEN
            DiagCode := 16#C003;
        ELSIF RTRIGatResetQ AND NOT NoExternalTest THEN
            DiagCode := 16#8004;
        ELSIF SOSSDIn AND (RTRIGatResetQ AND NoExternalTest) THEN
            DiagCode := 16#8010;
        END_IF;
    16#C020:
        IF Reset AND NOT RTRIGatResetQ THEN
            DiagCode := 16#C004;
        ELSIF RTRIGatResetQ AND NOT NoExternalTest THEN
            DiagCode := 16#8004;
        ELSIF SOSSDIn AND (RTRIGatResetQ AND NoExternalTest) THEN
            DiagCode := 16#8010;
        END_IF;
    END_CASE;
END_IF;
CASE DiagCode OF
16#0000:
    Ready := FALSE;
    SOSSDOut := FALSE;
    STestOut := TRUE;
    TestPossible := FALSE;
    TestExecuted := FALSE;
    Error := FALSE;
16#8000:
    Ready := TRUE;
    SOSSDOut := TRUE;
    STestOut := TRUE;
    TestPossible := TRUE;
    TestExecuted := TRUE;
    Error := FALSE;
16#8001, 16#8002, 16#8003, 16#8004, 16#8005, 16#8006:
    Ready := TRUE;
    SOSSDOut := FALSE;
    STestOut := TRUE;
    TestPossible := FALSE;
    TestExecuted := FALSE;
    Error := FALSE;
16#8010:
    Ready := TRUE;
    SOSSDOut := TRUE;
    STestOut := TRUE;
    TestPossible := TRUE;
    TestExecuted := FALSE;
    Error := FALSE;
16#8012, 16#8013:
    Ready := TRUE;
    SOSSDOut := FALSE;
    STestOut := TRUE;
    TestPossible := FALSE;
    TestExecuted := TRUE;
    Error := FALSE;
16#8020:
    Ready := TRUE;
    SOSSDOut := TRUE;
    STestOut := FALSE;
    TestPossible := FALSE;
    TestExecuted := FALSE;
    Error := FALSE;
    IN1:=TRUE;
    PT1:=TestTime;
    IF NOT running1 AND NOT Q1 THEN
        running1 := TRUE;
    ELSIF running1 AND NOT Q1 THEN
        Q1 := NONDETERMINISTIC_BOOL();
        running1 := NOT Q1;
    END_IF;
16#8030:
    Ready := TRUE;
    SOSSDOut := TRUE;
    STestOut := TRUE;
    TestPossible := FALSE;
    TestExecuted := FALSE;
    Error := FALSE;
    IN2:=TRUE;
    PT2:=TestTime;
    IF NOT running2 AND NOT Q2 THEN
        running2 := TRUE;
    ELSIF running2 AND NOT Q2 THEN
        Q2 := NONDETERMINISTIC_BOOL();
        running2 := NOT Q2;
    END_IF;
16#C000, 16#C001, 16#C002, 16#C003, 16#C004, 16#C005, 16#C006, 16#C010, 16#C020:
    Ready := TRUE;
    SOSSDOut := FALSE;
    STestOut := TRUE;
    TestPossible := FALSE;
    TestExecuted := FALSE;
    Error := TRUE;
16#C007:
    Ready := TRUE;
    SOSSDOut := FALSE;
    STestOut := TRUE;
    TestPossible := FALSE;
    TestExecuted := TRUE;
    Error := TRUE;
END_CASE;
END_FUNCTION_BLOCK

(* ---- SFTestableSafetySensor_CAP.st ---- *)
PROGRAM Main
VAR_INPUT
    Activate : BOOL;
    SOSSDIn : SAFEBOOL;
    StartTest : BOOL;
    TestTime : TIME := T#10ms;
    NoExternalTest : BOOL;
    SStartReset : SAFEBOOL;
    SAutoReset : SAFEBOOL;
    Reset : BOOL;
END_VAR
VAR
    SFTestableSafetySensor : SFTestableSafetySensor;
END_VAR
SFTestableSafetySensor(Activate:=Activate,SOSSDIn:=SOSSDIn,StartTest:=StartTest,TestTime:=TestTime,NoExternalTest:=NoExternalTest,
SStartReset:=SStartReset,SAutoReset:=SAutoReset,Reset:=Reset);
END_PROGRAM

FUNCTION_BLOCK SFTestableSafetySensor
VAR_INPUT
    Activate : BOOL;
    SOSSDIn : SAFEBOOL;
    StartTest : BOOL;
    TestTime : TIME := T#10ms;
    NoExternalTest : BOOL;
    SStartReset : SAFEBOOL;
    SAutoReset : SAFEBOOL;
    Reset : BOOL;
END_VAR
VAR
    IN1 : BOOL;
    PT1 : TIME;
    running1 : BOOL;
    Q1 : BOOL;
    IN2 : BOOL;
    PT2 : TIME;
    running2 : BOOL;
    Q2 : BOOL;
    RTRIGatResetQ : BOOL;
    RTRIGatResetM : BOOL;
    RTRIGatStartTestQ : BOOL;
    RTRIGatStartTestM : BOOL;
    FTRIGatSOSSDInQ : BOOL;
    FTRIGatSOSSDInM : BOOL;
END_VAR
VAR_OUTPUT
    Ready : SAFEBOOL;
    SOSSDOut : SAFEBOOL;
    STestOut : SAFEBOOL := TRUE;
    TestPossible : BOOL;
    TestExecuted : BOOL;
    Error : BOOL;
    DiagCode : WORD := 16#0000;
END_VAR
RTRIGatResetQ := Reset AND NOT RTRIGatResetM;
RTRIGatResetM := Reset;

RTRIGatStartTestQ := StartTest AND NOT RTRIGatStartTestM;
RTRIGatStartTestM := StartTest;

FTRIGatSOSSDInQ := NOT SOSSDIn AND FTRIGatSOSSDInM;
FTRIGatSOSSDInM := SOSSDIn;

IF NOT Activate THEN
    DiagCode := 16#0000;
ELSE
    CASE DiagCode OF
    16#0000:
        IF Activate THEN
            DiagCode := 16#8001;
        END_IF;
    16#8000:
        IF NOT SOSSDIn THEN
            DiagCode := 16#8012;
        ELSIF RTRIGatStartTestQ THEN
            DiagCode := 16#8020;
            IN1:=FALSE;
            Q1 := FALSE;
            running1 := FALSE;
        END_IF;
    16#8001:
        IF TestTime > T#150ms THEN
            DiagCode := 16#C000;
        ELSIF Reset AND NOT RTRIGatResetQ AND NOT SStartReset THEN
            DiagCode := 16#C001;
        ELSIF NOT SOSSDIn THEN
            DiagCode := 16#8002;
        ELSIF SOSSDIn AND (RTRIGatResetQ OR SStartReset) THEN
            DiagCode := 16#8010;
        END_IF;
    16#8002:
        IF SOSSDIn THEN
            DiagCode := 16#8003;
        END_IF;
    16#8003:
        IF Reset AND NOT RTRIGatResetQ AND NOT SAutoReset THEN
            DiagCode := 16#C002;
        ELSIF NOT SOSSDIn THEN
            DiagCode := 16#8002;
        ELSIF SOSSDIn AND (RTRIGatResetQ OR SAutoReset) THEN
            DiagCode := 16#8010;
        END_IF;
    16#8004:
        IF FTRIGatSOSSDInQ THEN
            DiagCode := 16#8005;
        END_IF;
    16#8005:
        IF SOSSDIn THEN
            DiagCode := 16#8006;
        END_IF;
    16#8006:
        IF Reset AND NOT RTRIGatResetQ THEN
            DiagCode := 16#C005;
        ELSIF RTRIGatResetQ AND NOT SOSSDIn THEN
            DiagCode := 16#8002;
        ELSIF RTRIGatResetQ AND SOSSDIn THEN
            DiagCode := 16#8010;
        END_IF;
    16#8010:
        IF NOT SOSSDIn THEN
            DiagCode := 16#8002;
        ELSIF RTRIGatStartTestQ THEN
            DiagCode := change(16#8020, 16#8002);
            IN1:=FALSE;
            Q1 := FALSE;
            running1 := FALSE;
        END_IF;
    16#8012:
        IF SOSSDIn THEN
            DiagCode := 16#8013;
        END_IF;
    16#8013:
        IF Reset AND NOT RTRIGatResetQ AND NOT SAutoReset THEN
            DiagCode := 16#C007;
        ELSIF NOT SOSSDIn THEN
            DiagCode := 16#8012;
        ELSIF SOSSDIn AND (RTRIGatResetQ OR SAutoReset) THEN
            DiagCode := 16#8000;
        END_IF;
    16#8020:
        IF Q1 THEN
            DiagCode := 16#C020;
        ELSIF NOT SOSSDIn THEN
            DiagCode := 16#8030;
            IN2:=FALSE;
            Q2 := FALSE;
            running2 := FALSE;
        END_IF;
    16#8030:
        IF Q2 THEN
            DiagCode := 16#C030;
        ELSIF SOSSDIn THEN
            DiagCode := 16#8000;
        END_IF;
    16#C000:
        IF Reset AND NOT RTRIGatResetQ THEN
            DiagCode := 16#C006;
        ELSIF RTRIGatResetQ AND TestTime <= T#150ms THEN
            DiagCode := 16#8001;
        END_IF;
    16#C001:
        IF NOT Reset THEN
            DiagCode := 16#8001;
        END_IF;
    16#C002:
        IF NOT Reset THEN
            DiagCode := 16#8003;
        END_IF;
    16#C003:
        IF NOT Reset THEN
            DiagCode := 16#C010;
        END_IF;
    16#C004:
        IF NOT Reset THEN
            DiagCode := 16#C020;
        END_IF;
    16#C005:
        IF NOT Reset THEN
            DiagCode := 16#8006;
        END_IF;
    16#C006:
        IF NOT Reset THEN
            DiagCode := 16#C000;
        END_IF;
    16#C007:
        IF NOT Reset THEN
            DiagCode := 16#8013;
        END_IF;
    16#C010:
        IF Reset AND NOT RTRIGatResetQ THEN
            DiagCode := 16#C003;
        ELSIF RTRIGatResetQ AND NOT NoExternalTest THEN
            DiagCode := 16#8004;
        ELSIF SOSSDIn AND (RTRIGatResetQ AND NoExternalTest) THEN
            DiagCode := 16#8010;
        END_IF;
    16#C020:
        IF Reset AND NOT RTRIGatResetQ THEN
            DiagCode := 16#C004;
        ELSIF RTRIGatResetQ AND NOT NoExternalTest THEN
            DiagCode := 16#8004;
        ELSIF SOSSDIn AND (RTRIGatResetQ AND NoExternalTest) THEN
            DiagCode := 16#8010;
        END_IF;
    END_CASE;
END_IF;
CASE DiagCode OF
16#0000:
    Ready := FALSE;
    SOSSDOut := FALSE;
    STestOut := TRUE;
    TestPossible := FALSE;
    TestExecuted := FALSE;
    Error := FALSE;
16#8000:
    Ready := TRUE;
    SOSSDOut := TRUE;
    STestOut := TRUE;
    TestPossible := TRUE;
    TestExecuted := TRUE;
    Error := FALSE;
16#8001, 16#8002, 16#8003, 16#8004, 16#8005, 16#8006:
    Ready := TRUE;
    SOSSDOut := FALSE;
    STestOut := TRUE;
    TestPossible := FALSE;
    TestExecuted := FALSE;
    Error := FALSE;
16#8010:
    Ready := TRUE;
    SOSSDOut := TRUE;
    STestOut := TRUE;
    TestPossible := TRUE;
    TestExecuted := FALSE;
    Error := FALSE;
16#8012, 16#8013:
    Ready := TRUE;
    SOSSDOut := FALSE;
    STestOut := TRUE;
    TestPossible := FALSE;
    TestExecuted := TRUE;
    Error := FALSE;
16#8020:
    Ready := TRUE;
    SOSSDOut := TRUE;
    STestOut := FALSE;
    TestPossible := FALSE;
    TestExecuted := FALSE;
    Error := FALSE;
    IN1:=TRUE;
    PT1:=TestTime;
    IF NOT running1 AND NOT Q1 THEN
        running1 := TRUE;
    ELSIF running1 AND NOT Q1 THEN
        Q1 := NONDETERMINISTIC_BOOL();
        running1 := NOT Q1;
    END_IF;
16#8030:
    Ready := TRUE;
    SOSSDOut := TRUE;
    STestOut := TRUE;
    TestPossible := FALSE;
    TestExecuted := FALSE;
    Error := FALSE;
    IN2:=TRUE;
    PT2:=TestTime;
    IF NOT running2 AND NOT Q2 THEN
        running2 := TRUE;
    ELSIF running2 AND NOT Q2 THEN
        Q2 := NONDETERMINISTIC_BOOL();
        running2 := NOT Q2;
    END_IF;
16#C000, 16#C001, 16#C002, 16#C003, 16#C004, 16#C005, 16#C006, 16#C010, 16#C020:
    Ready := TRUE;
    SOSSDOut := FALSE;
    STestOut := TRUE;
    TestPossible := FALSE;
    TestExecuted := FALSE;
    Error := TRUE;
16#C007:
    Ready := TRUE;
    SOSSDOut := FALSE;
    STestOut := TRUE;
    TestPossible := FALSE;
    TestExecuted := TRUE;
    Error := TRUE;
END_CASE;
END_FUNCTION_BLOCK

(* ---- SFTwoHandControlTypeII.st ---- *)
PROGRAM Main
VAR_INPUT
    Activate : BOOL;
    SButton1 : SAFEBOOL;
    SButton2 : SAFEBOOL;
END_VAR
VAR
    SFTwoHandControlTypeII : SFTwoHandControlTypeII;
END_VAR
SFTwoHandControlTypeII(Activate:=Activate,SButton1:=SButton1,SButton2:=SButton2);
END_PROGRAM

FUNCTION_BLOCK SFTwoHandControlTypeII
VAR_INPUT
    Activate : BOOL;
    SButton1 : SAFEBOOL;
    SButton2 : SAFEBOOL;
END_VAR
VAR_OUTPUT
    Ready : BOOL;
    STwoHandOut : BOOL;
    Error : BOOL;
    DiagCode : WORD;
END_VAR
IF NOT Activate THEN
    DiagCode := 16#0000;
ELSE
    CASE DiagCode OF
    16#0000:
        IF Activate THEN
            DiagCode := 16#8001;
        END_IF;
    16#8001:
        IF SButton1 AND SButton2 THEN
            DiagCode := 16#C003;
        ELSIF SButton1 THEN
            DiagCode := 16#C001;
        ELSIF SButton2 THEN
            DiagCode := 16#C002;
        ELSE
            DiagCode := 16#8004;
        END_IF;
    16#8004:
        IF SButton1 AND SButton2 THEN
            DiagCode := 16#8000;
        ELSIF SButton1 THEN
            DiagCode := 16#8005;
        ELSIF SButton2 THEN
            DiagCode := 16#8006;
        END_IF;
    16#8005:
        IF NOT (SButton1 OR SButton2) THEN
            DiagCode := 16#8004;
        ELSIF NOT SButton1 AND SButton2 THEN
            DiagCode := 16#8019;
        ELSIF SButton1 AND SButton2 THEN
            DiagCode := 16#8000;
        END_IF;
    16#8006:
        IF NOT (SButton1 OR SButton2) THEN
            DiagCode := 16#8004;
        ELSIF SButton1 AND NOT SButton2 THEN
            DiagCode := 16#8019;
        ELSIF SButton1 AND SButton2 THEN
            DiagCode := 16#8000;
        END_IF;
    16#8007:
        IF SButton1 AND SButton2 THEN
            DiagCode := 16#8009;
        ELSIF NOT SButton1 AND SButton2 THEN
            DiagCode := 16#8008;
        ELSIF NOT (SButton1 OR SButton2) THEN
            DiagCode := 16#8004;
        END_IF;
    16#8008:
        IF SButton1 AND SButton2 THEN
            DiagCode := 16#8009;
        ELSIF SButton1 AND NOT SButton2 THEN
            DiagCode := 16#8007;
        ELSIF NOT (SButton1 OR SButton2) THEN
            DiagCode := 16#8004;
        END_IF;
    16#8009:
        IF NOT SButton1 AND SButton2 THEN
            DiagCode := 16#8008;
        ELSIF SButton1 AND NOT SButton2 THEN
            DiagCode := 16#8007;
        ELSIF NOT (SButton1 OR SButton2) THEN
            DiagCode := 16#8004;
        END_IF;
    16#8019:
        IF NOT (SButton1 OR SButton2) THEN
            DiagCode := 16#8004;
        END_IF;
    16#8000:
        IF SButton1 AND NOT SButton2 THEN
            DiagCode := 16#8007;
        ELSIF NOT SButton1 AND SButton2 THEN
            DiagCode := 16#8008;
        ELSIF NOT (SButton1 OR SButton2) THEN
            DiagCode := 16#8004;
        END_IF;
    16#C001,
    16#C002,
    16#C003:
        IF NOT (SButton1 OR SButton2) THEN
            DiagCode := 16#8004;
        END_IF;
    END_CASE;
END_IF;
CASE DiagCode OF
16#0000:
    Ready := FALSE;
    Error := FALSE;
    STwoHandOut := FALSE;
16#8000:
    Ready := TRUE;
    Error := FALSE;
    STwoHandOut := TRUE;
16#8001,
16#8004,
16#8005,
16#8006,
16#8007,
16#8008,
16#8009,
16#8019:
    Ready := TRUE;
    Error := FALSE;
    STwoHandOut := FALSE;
16#C001,
16#C002,
16#C003:
    Ready := TRUE;
    Error := TRUE;
    STwoHandOut := FALSE;
END_CASE;
END_FUNCTION_BLOCK

(* ---- SFTwoHandControlTypeII_CAP.st ---- *)
PROGRAM Main
VAR_INPUT
    Activate : BOOL;
    SButton1 : SAFEBOOL;
    SButton2 : SAFEBOOL;
END_VAR
VAR
    SFTwoHandControlTypeII : SFTwoHandControlTypeII;
END_VAR
SFTwoHandControlTypeII(Activate:=Activate,SButton1:=SButton1,SButton2:=SButton2);
END_PROGRAM

FUNCTION_BLOCK SFTwoHandControlTypeII
VAR_INPUT
    Activate : BOOL;
    SButton1 : SAFEBOOL;
    SButton2 : SAFEBOOL;
END_VAR
VAR_OUTPUT
    Ready : BOOL;
    STwoHandOut : BOOL;
    Error : BOOL;
    DiagCode : WORD;
END_VAR
IF NOT Activate THEN
    DiagCode := 16#0000;
ELSE
    CASE DiagCode OF
    16#0000:
        IF Activate THEN
            DiagCode := 16#8001;
        END_IF;
    16#8001:
        IF SButton1 AND SButton2 THEN
            DiagCode := 16#C003;
        ELSIF SButton1 THEN
            DiagCode := 16#C001;
        ELSIF SButton2 THEN
            DiagCode := 16#C002;
        ELSE
            DiagCode := 16#8004;
        END_IF;
    16#8004:
        IF SButton1 AND SButton2 THEN
            DiagCode := 16#8000;
        ELSIF SButton1 THEN
            DiagCode := 16#8005;
        ELSIF SButton2 THEN
            DiagCode := 16#8006;
        END_IF;
    16#8005:
        IF NOT (SButton1 OR SButton2) THEN
            DiagCode := 16#8004;
        ELSIF NOT SButton1 AND SButton2 THEN
            DiagCode := 16#8019;
        ELSIF SButton1 AND SButton2 THEN
            DiagCode := 16#8000;
        END_IF;
    16#8006:
        IF NOT (SButton1 OR SButton2) THEN
            DiagCode := 16#8004;
        ELSIF SButton1 AND NOT SButton2 THEN
            DiagCode := 16#8019;
        ELSIF SButton1 AND SButton2 THEN
            DiagCode := 16#8000;
        END_IF;
    16#8007:
        IF SButton1 AND SButton2 THEN
            DiagCode := 16#8009;
        ELSIF NOT SButton1 AND SButton2 THEN
            DiagCode := 16#8008;
        ELSIF NOT (SButton1 OR SButton2) THEN
            DiagCode := 16#8004;
        END_IF;
    16#8008:
        IF SButton1 AND SButton2 THEN
            DiagCode := 16#8009;
        ELSIF SButton1 AND NOT SButton2 THEN
            DiagCode := 16#8007;
        ELSIF NOT (SButton1 OR SButton2) THEN
            DiagCode := 16#8004;
        END_IF;
    16#8009:
        IF NOT SButton1 AND SButton2 THEN
            DiagCode := change(16#8008, 16#8007);
        ELSIF SButton1 AND NOT SButton2 THEN
            DiagCode := 16#8007;
        ELSIF NOT (SButton1 OR SButton2) THEN
            DiagCode := 16#8004;
        END_IF;
    16#8019:
        IF NOT (SButton1 OR SButton2) THEN
            DiagCode := 16#8004;
        END_IF;
    16#8000:
        IF SButton1 AND NOT SButton2 THEN
            DiagCode := 16#8007;
        ELSIF NOT SButton1 AND SButton2 THEN
            DiagCode := 16#8008;
        ELSIF NOT (SButton1 OR SButton2) THEN
            DiagCode := 16#8004;
        END_IF;
    16#C001,
    16#C002,
    16#C003:
        IF NOT (SButton1 OR SButton2) THEN
            DiagCode := 16#8004;
        END_IF;
    END_CASE;
END_IF;
CASE DiagCode OF
16#0000:
    Ready := FALSE;
    Error := FALSE;
    STwoHandOut := FALSE;
16#8000:
    Ready := TRUE;
    Error := FALSE;
    STwoHandOut := TRUE;
16#8001,
16#8004,
16#8005,
16#8006,
16#8007,
16#8008,
16#8009,
16#8019:
    Ready := TRUE;
    Error := FALSE;
    STwoHandOut := FALSE;
16#C001,
16#C002,
16#C003:
    Ready := TRUE;
    Error := TRUE;
    STwoHandOut := FALSE;
END_CASE;
END_FUNCTION_BLOCK

(* ---- SFTwoHandControlTypeIII.st ---- *)
PROGRAM Main
VAR_INPUT
    Activate : BOOL;
    SButton1 : SAFEBOOL;
    SButton2 : SAFEBOOL;
END_VAR
VAR
    SFTwoHandControlTypeIII : SFTwoHandControlTypeIII;
END_VAR
SFTwoHandControlTypeIII(Activate:=Activate,SButton1:=SButton1,SButton2:=SButton2);
END_PROGRAM

FUNCTION_BLOCK SFTwoHandControlTypeIII
VAR_INPUT
    Activate : BOOL;
    SButton1 : SAFEBOOL;
    SButton2 : SAFEBOOL;
END_VAR
VAR
    IN : BOOL;
    PT : TIME;
    running : BOOL;
    Q : BOOL;
END_VAR
VAR_OUTPUT
    Ready : BOOL;
    STwoHandOut : SAFEBOOL;
    Error : BOOL;
    DiagCode : WORD:=16#0000;
END_VAR
IF NOT Activate THEN
    DiagCode := 16#0000;
ELSE
    CASE DiagCode OF
    16#0000:
        IF Activate THEN
            DiagCode := 16#8001;
        END_IF;
    16#8000:
        IF SButton1 AND NOT SButton2 THEN
            DiagCode := 16#8007;
        ELSIF NOT SButton1 AND SButton2 THEN
            DiagCode := 16#8008;
        ELSIF NOT (SButton1 OR SButton2) THEN
            DiagCode := 16#8004;
        END_IF;
    16#8001:
        IF SButton1 AND SButton2 THEN
            DiagCode := 16#C003;
        ELSIF SButton1 THEN
            DiagCode := 16#C001;
        ELSIF SButton2 THEN
            DiagCode := 16#C002;
        ELSIF NOT (SButton1 OR SButton2) THEN
            DiagCode := 16#8004;
        END_IF;
    16#8004:
        IF SButton1 AND SButton2 THEN
            DiagCode := 16#8000;
        ELSIF SButton1 THEN
            DiagCode := 16#8005;
        ELSIF SButton2 THEN
            DiagCode := 16#8006;
        END_IF;
    16#8005:
        IF Q THEN
            IF SButton1 AND SButton2 THEN
                DiagCode := 16#C006;
            ELSIF SButton1 THEN
                DiagCode := 16#C005;
            ELSIF SButton2 THEN
                DiagCode := 16#C004;
            END_IF;
        ELSIF NOT (SButton1 OR SButton2) THEN
            DiagCode := 16#8004;
        ELSIF NOT SButton1 AND SButton2 THEN
            DiagCode := 16#8019;
        ELSIF SButton1 AND SButton2 THEN
            DiagCode := 16#8000;
        END_IF;
    16#8006:
        IF Q THEN
            IF SButton1 AND SButton2 THEN
                DiagCode := 16#C006;
            ELSIF SButton1 THEN
                DiagCode := 16#C005;
            ELSIF SButton2 THEN
                DiagCode := 16#C004;
            END_IF;
        ELSIF NOT (SButton1 OR SButton2) THEN
            DiagCode := 16#8004;
        ELSIF SButton1 AND NOT SButton2 THEN
            DiagCode := 16#8019;
        ELSIF SButton1 AND SButton2 THEN
            DiagCode := 16#8000;
        END_IF;
    16#8007:
        IF SButton1 AND SButton2 THEN
            DiagCode := 16#8009;
        ELSIF NOT SButton1 AND SButton2 THEN
            DiagCode := 16#8008;
        ELSIF NOT (SButton1 OR SButton2) THEN
            DiagCode := 16#8004;
        END_IF;
    16#8008:
        IF SButton1 AND SButton2 THEN
            DiagCode := 16#8009;
        ELSIF SButton1 AND NOT SButton2 THEN
            DiagCode := 16#8007;
        ELSIF NOT (SButton1 OR SButton2) THEN
            DiagCode := 16#8004;
        END_IF;
    16#8009:
        IF NOT SButton1 AND SButton2 THEN
            DiagCode := 16#8008;
        ELSIF SButton1 AND NOT SButton2 THEN
            DiagCode := 16#8007;
        ELSIF NOT (SButton1 OR SButton2) THEN
            DiagCode := 16#8004;
        END_IF;
    16#8019:
        IF NOT (SButton1 OR SButton2) THEN
            DiagCode := 16#8004;
        END_IF;
    16#C001,
    16#C002,
    16#C003,
    16#C004,
    16#C005,
    16#C006:
        IF NOT (SButton1 OR SButton2) THEN
            DiagCode := 16#8004;
        END_IF;
    END_CASE;
END_IF;
IF DiagCode = 16#8005 OR DiagCode = 16#8006 THEN
    IN:=TRUE;
    PT:=TIME#500ms;
    IF NOT running AND NOT Q THEN
        running := TRUE;
    ELSIF running AND NOT Q THEN
        Q := NONDETERMINISTIC_BOOL();
        running := NOT Q;
    END_IF;
ELSE
    IN:=FALSE;
    PT:=TIME#500ms;
    Q := FALSE;
    running := FALSE;
END_IF;
CASE DiagCode OF
16#0000:
    Ready := FALSE;
    STwoHandOut := FALSE;
    Error := FALSE;
16#8000:
    Ready := TRUE;
    STwoHandOut := TRUE;
    Error := FALSE;
16#8001,
16#8004,
16#8005,
16#8006,
16#8007,
16#8008,
16#8009,
16#8019:
    Ready := TRUE;
    STwoHandOut := FALSE;
    Error := FALSE;
16#C001,
16#C002,
16#C003,
16#C004,
16#C005,
16#C006:
    Ready := TRUE;
    STwoHandOut := FALSE;
    Error := TRUE;
END_CASE;
END_FUNCTION_BLOCK

(* ---- SFTwoHandControlTypeIII_CAP.st ---- *)
PROGRAM Main
VAR_INPUT
    Activate : BOOL;
    SButton1 : SAFEBOOL;
    SButton2 : SAFEBOOL;
END_VAR
VAR
    SFTwoHandControlTypeIII : SFTwoHandControlTypeIII;
END_VAR
SFTwoHandControlTypeIII(Activate:=Activate,SButton1:=SButton1,SButton2:=SButton2);
END_PROGRAM

FUNCTION_BLOCK SFTwoHandControlTypeIII
VAR_INPUT
    Activate : BOOL;
    SButton1 : SAFEBOOL;
    SButton2 : SAFEBOOL;
END_VAR
VAR
    IN : BOOL;
    PT : TIME;
    running : BOOL;
    Q : BOOL;
END_VAR
VAR_OUTPUT
    Ready : BOOL;
    STwoHandOut : SAFEBOOL;
    Error : BOOL;
    DiagCode : WORD:=16#0000;
END_VAR
IF NOT Activate THEN
    DiagCode := 16#0000;
ELSE
    CASE DiagCode OF
    16#0000:
        IF Activate THEN
            DiagCode := 16#8001;
        END_IF;
    16#8000:
        IF SButton1 AND NOT SButton2 THEN
            DiagCode := 16#8007;
        ELSIF NOT SButton1 AND SButton2 THEN
            DiagCode := 16#8008;
        ELSIF NOT (SButton1 OR SButton2) THEN
            DiagCode := 16#8004;
        END_IF;
    16#8001:
        IF SButton1 AND SButton2 THEN
            DiagCode := 16#C003;
        ELSIF SButton1 THEN
            DiagCode := 16#C001;
        ELSIF SButton2 THEN
            DiagCode := 16#C002;
        ELSIF NOT (SButton1 OR SButton2) THEN
            DiagCode := 16#8004;
        END_IF;
    16#8004:
        IF SButton1 AND SButton2 THEN
            DiagCode := 16#8000;
        ELSIF SButton1 THEN
            DiagCode := change(16#8005, 16#8000);
        ELSIF SButton2 THEN
            DiagCode := 16#8006;
        END_IF;
    16#8005:
        IF Q THEN
            IF SButton1 AND SButton2 THEN
                DiagCode := 16#C006;
            ELSIF SButton1 THEN
                DiagCode := 16#C005;
            ELSIF SButton2 THEN
                DiagCode := 16#C004;
            END_IF;
        ELSIF NOT (SButton1 OR SButton2) THEN
            DiagCode := 16#8004;
        ELSIF NOT SButton1 AND SButton2 THEN
            DiagCode := 16#8019;
        ELSIF SButton1 AND SButton2 THEN
            DiagCode := 16#8000;
        END_IF;
    16#8006:
        IF Q THEN
            IF SButton1 AND SButton2 THEN
                DiagCode := 16#C006;
            ELSIF SButton1 THEN
                DiagCode := 16#C005;
            ELSIF SButton2 THEN
                DiagCode := 16#C004;
            END_IF;
        ELSIF NOT (SButton1 OR SButton2) THEN
            DiagCode := 16#8004;
        ELSIF SButton1 AND NOT SButton2 THEN
            DiagCode := 16#8019;
        ELSIF SButton1 AND SButton2 THEN
            DiagCode := 16#8000;
        END_IF;
    16#8007:
        IF SButton1 AND SButton2 THEN
            DiagCode := 16#8009;
        ELSIF NOT SButton1 AND SButton2 THEN
            DiagCode := 16#8008;
        ELSIF NOT (SButton1 OR SButton2) THEN
            DiagCode := 16#8004;
        END_IF;
    16#8008:
        IF SButton1 AND SButton2 THEN
            DiagCode := 16#8009;
        ELSIF SButton1 AND NOT SButton2 THEN
            DiagCode := 16#8007;
        ELSIF NOT (SButton1 OR SButton2) THEN
            DiagCode := 16#8004;
        END_IF;
    16#8009:
        IF NOT SButton1 AND SButton2 THEN
            DiagCode := 16#8008;
        ELSIF SButton1 AND NOT SButton2 THEN
            DiagCode := 16#8007;
        ELSIF NOT (SButton1 OR SButton2) THEN
            DiagCode := 16#8004;
        END_IF;
    16#8019:
        IF NOT (SButton1 OR SButton2) THEN
            DiagCode := 16#8004;
        END_IF;
    16#C001,
    16#C002,
    16#C003,
    16#C004,
    16#C005,
    16#C006:
        IF NOT (SButton1 OR SButton2) THEN
            DiagCode := 16#8004;
        END_IF;
    END_CASE;
END_IF;
IF DiagCode = 16#8005 OR DiagCode = 16#8006 THEN
    IN:=TRUE;
    PT:=TIME#500ms;
    IF NOT running AND NOT Q THEN
        running := TRUE;
    ELSIF running AND NOT Q THEN
        Q := NONDETERMINISTIC_BOOL();
        running := NOT Q;
    END_IF;
ELSE
    IN:=FALSE;
    PT:=TIME#500ms;
    Q := FALSE;
    running := FALSE;
END_IF;
CASE DiagCode OF
16#0000:
    Ready := FALSE;
    STwoHandOut := FALSE;
    Error := FALSE;
16#8000:
    Ready := TRUE;
    STwoHandOut := TRUE;
    Error := FALSE;
16#8001,
16#8004,
16#8005,
16#8006,
16#8007,
16#8008,
16#8009,
16#8019:
    Ready := TRUE;
    STwoHandOut := FALSE;
    Error := FALSE;
16#C001,
16#C002,
16#C003,
16#C004,
16#C005,
16#C006:
    Ready := TRUE;
    STwoHandOut := FALSE;
    Error := TRUE;
END_CASE;
END_FUNCTION_BLOCK
